# EPICS autosave request: iocBoot/iocEnergy_2BM/auto_settings.req
file "energy_settings.req", P=$(P), R=$(R)
